{attribute 'GeneratedUsingTerminal: EL5151-0090-0016'}
{attribute addProperty BoxType "EL5151-0090-0016"}
{attribute addProperty Id "ENC_Status_compactAT %I*ENC_Status_compact_B353648514ENC_Control_compactAT %Q*ENC_Control_compact_21E2D14D6WcStateAT %I*WcState_9091E0EB2InfoDataAT %I*InfoData_94A18F5E2"}
{attribute addProperty CRC "3904677945"}
{attribute addProperty Size "24"}
TYPE EL5151_E8BCA839 EXTENDS EtcSlaveTerminalBase_947E5A46 :
STRUCT
	{attribute addProperty Name "ENC_Status_compact"}
	ENC_Status_compact : ENC_Status_compact_B3536485;
	{attribute addProperty Name "ENC_Control_compact"}
	ENC_Control_compact : ENC_Control_compact_21E2D14D;
	{attribute addProperty Name "WcState"}
	WcState : WcState_9091E0EB;
	{attribute addProperty Name "InfoData"}
	InfoData : InfoData_94A18F5E;
END_STRUCT
END_TYPE

(* stored: Version 1.2.0.0, ProductVersion 3.1.4024.9
   DUT EL5151_E8BCA839: Id {c99f9e0c-d779-416a-8437-f4fc5a84aae5} *)
